{attribute 'GeneratedUsingTerminal: EP1859-0042-0018'}
{attribute addProperty BoxType "EP1859-0042-0018"}
{attribute addProperty Id "OutputAT %Q*BOOL1"}
{attribute addProperty CRC "1120571895"}
{attribute addProperty Size "1"}
TYPE DO_X05_Pin_42CA91F7 :
STRUCT
	{attribute addProperty Name "Output"}
	Output AT %Q* : BOOL;
END_STRUCT
END_TYPE

(* stored: Version 1.2.0.0, ProductVersion 3.1.4024.9
   DUT DO_X05_Pin_42CA91F7: Id {e2400afc-f000-442a-a89d-eb3a98bc1fdc} *)
